// SIMATIC S7-200 SMART project (STEP 7-Micro/WIN SMART), CPU ST40

SYMBOL_TABLE Table 1
Item_detected    V0.0
Lid_at_place     V0.1
Base_at_place    V0.2
Part_leaving     V0.3
Start            V0.4
Reset            V0.5
Stop_            V0.6
Emergency_stop   V0.7
Auto             V1.0
FACTORY_IO_Running V1.1
X                VD100
Z                VD104
Lids_conveyor_1  Q2.0     // 0
Stop_blade_1     Q0.1
Lids_conveyor_2  Q2.1     // 0
Bases_conveyor_1 Q2.2     // 0
Stop_blade_2     Q0.4
Bases_conveyor_2 Q2.3     // 0
Grab             Q0.6
Start_light      Q0.7
Reset_light      Q1.0
Stop_light       Q1.1
Step_1_light     Q1.2
Step_2_light     Q1.3
Step_3_light     Q1.4
FACTOR_IO_Reset  Q1.5
Set_X            QD4
Set_Z            QD8
Counter          QD12
END_SYMBOL_TABLE

SYMBOL_TABLE System Symbols
Always_On        SM0.0    // Always ON
END_SYMBOL_TABLE

ORGANIZATION_BLOCK MAIN:OB1
TITLE=Program Comments
BEGIN
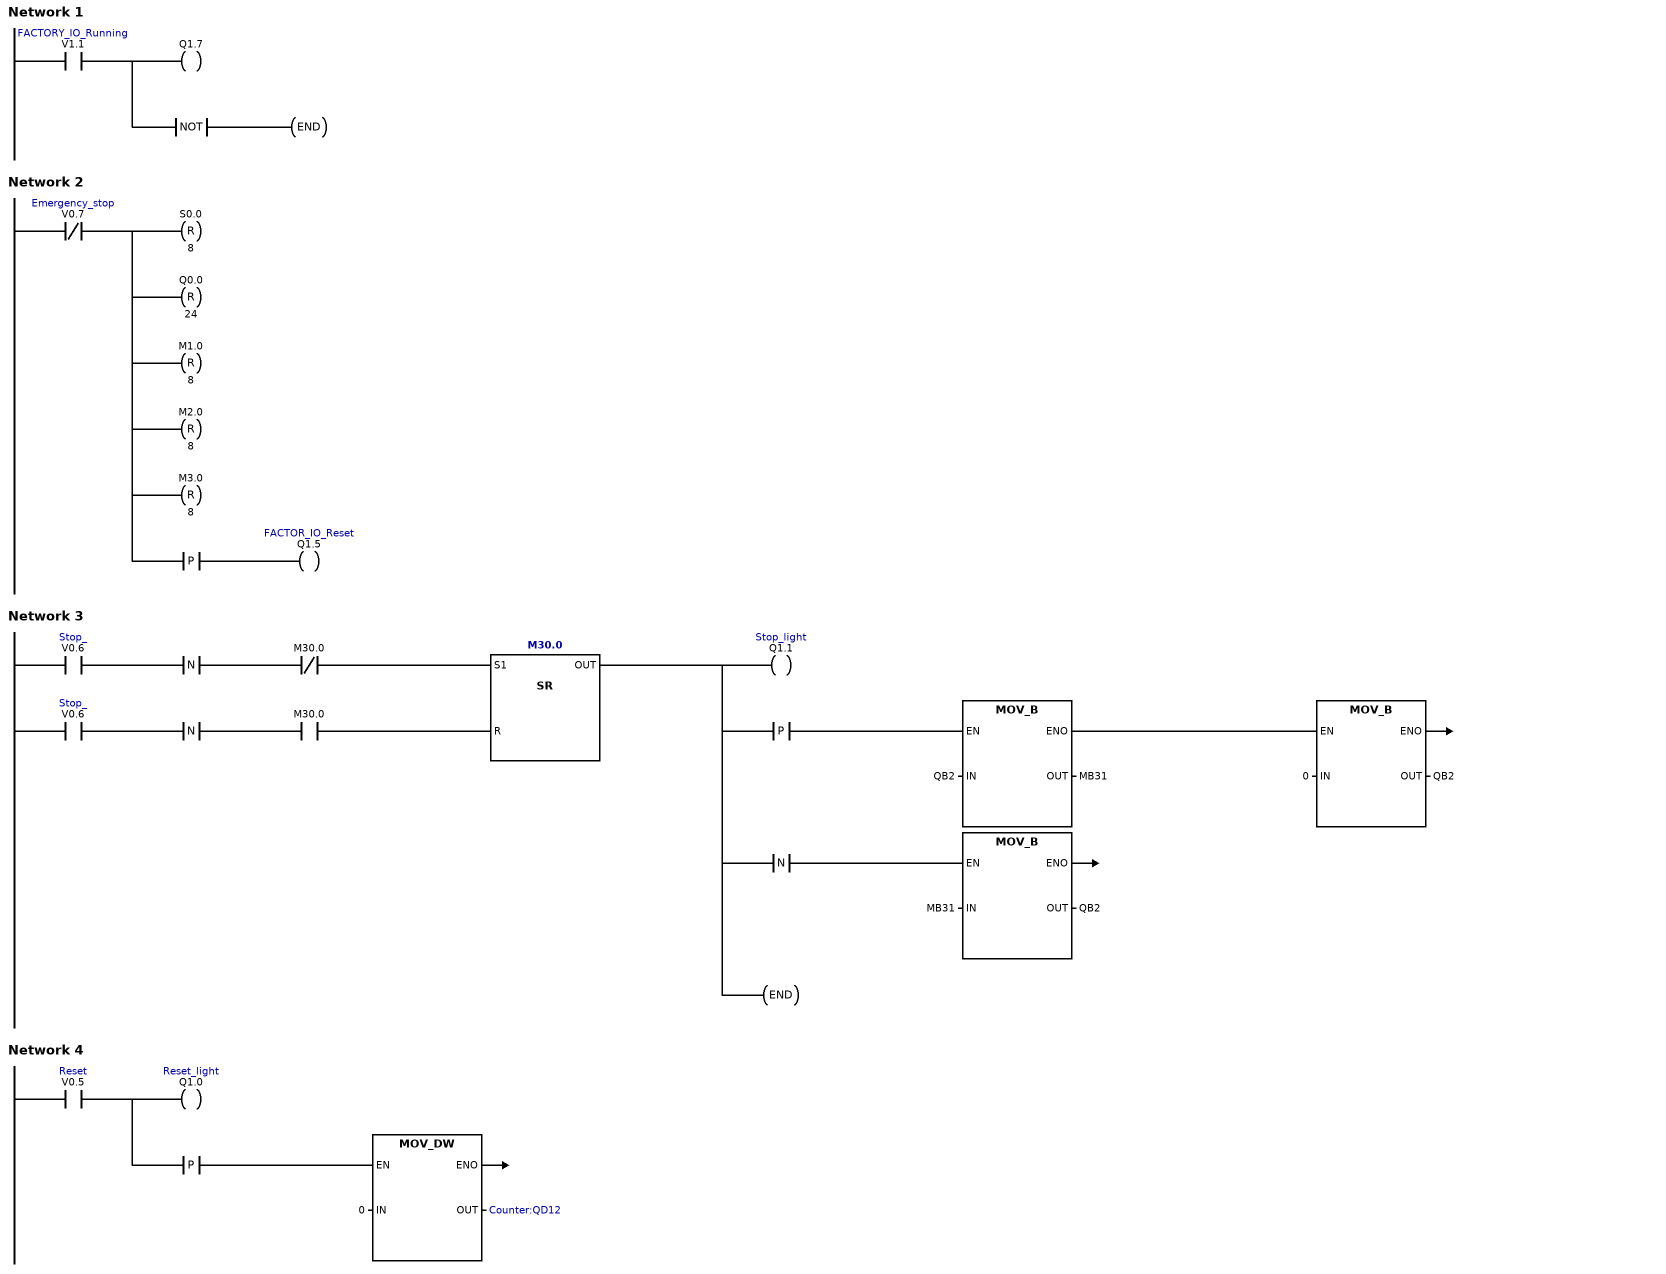
Network 1
LD     FACTORY_IO_Running:V1.1
=      Q1.7
NOT
END
Network 2
LDN    Emergency_stop:V0.7
R      S0.0, 8
R      Q0.0, 24
R      M1.0, 8
R      M2.0, 8
R      M3.0, 8
EU
=      FACTOR_IO_Reset:Q1.5
Network 3
LD     Stop_:V0.6
ED
AN     M30.0
LD     Stop_:V0.6
ED
A      M30.0
NOT
A      M30.0
OLD
=      M30.0
LPS
=      Stop_light:Q1.1
EU
MOVB   QB2, MB31
AENO
MOVB   0, QB2
LRD
ED
MOVB   MB31, QB2
LPP
END
Network 4
LD     Reset:V0.5
=      Reset_light:Q1.0
EU
MOVD   0, Counter:QD12
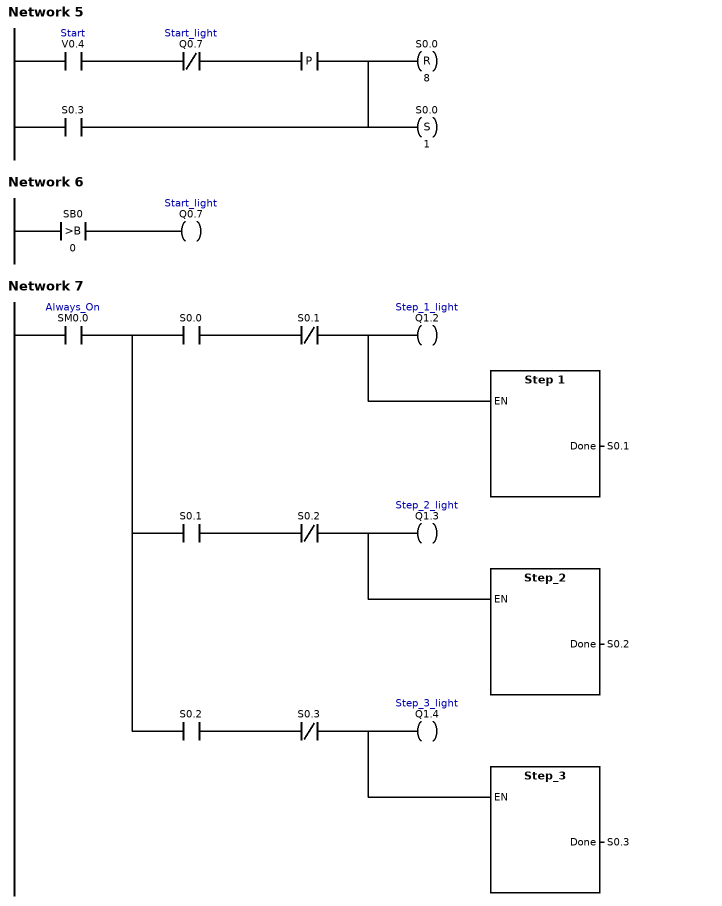
Network 5
LD     Start:V0.4
AN     Start_light:Q0.7
EU
O      S0.3
R      S0.0, 8
S      S0.0, 1
Network 6
LDB>   SB0, 0
=      Start_light:Q0.7
Network 7
LD     Always_On:SM0.0
LPS
A      S0.0
AN     S0.1
=      Step_1_light:Q1.2
CALL   Step 1:SBR1, S0.1
LRD
A      S0.1
AN     S0.2
=      Step_2_light:Q1.3
CALL   Step_2:SBR2, S0.2
LPP
A      S0.2
AN     S0.3
=      Step_3_light:Q1.4
CALL   Step_3:SBR3, S0.3
END_ORGANIZATION_BLOCK

SUBROUTINE_BLOCK Move:SBR0
TITLE=Subroutine Comments
VAR_INPUT
Set_X:REAL;	// LD0 
Set_Z:REAL;	// LD4 
END_VAR
VAR_OUTPUT
Done:BOOL;	// L8.0 
END_VAR
VAR
tmp:BOOL;	// L8.1 
tmp_x:REAL;	// LD9 
tmp_z:REAL;	// LD13 
END_VAR
BEGIN
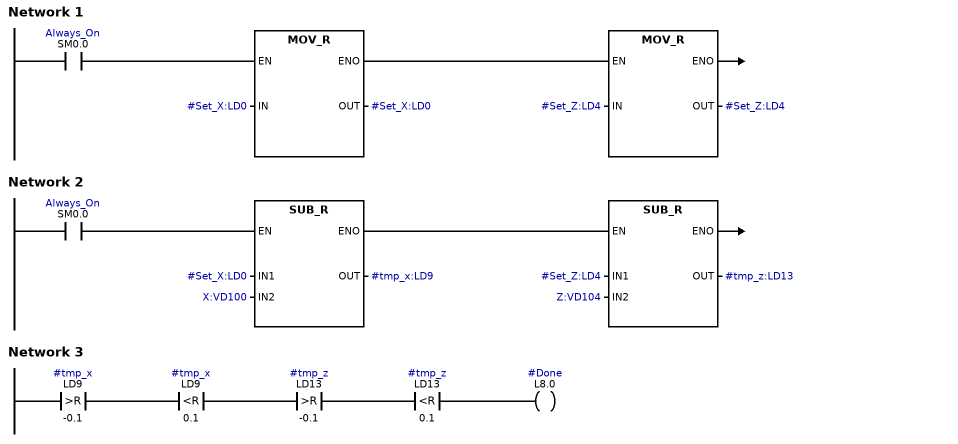
Network 1
LD     Always_On:SM0.0
MOVR   #Set_X:LD0, Set_X:QD4
AENO
MOVR   #Set_Z:LD4, Set_Z:QD8
Network 2
// (network saved uncompiled; LAD cells follow)
// row 0: c0 -| |- Always_On:SM0.0  c1 --  c2 [SUB_R EN:=power@row0, IN1:=#Set_X:LD0, IN2:=X:VD100, ENO=>power, OUT=>#tmp_x:LD9]  c3 --  c4 --  c5 [SUB_R EN:=power@row0, IN1:=#Set_Z:LD4, IN2:=Z:VD104, ENO=>power, OUT=>#tmp_z:LD13]  c6 ->
// row 1: c2 [box]  c5 [box]
Network 3
LDR>   #tmp_x:LD9, -0.1
AR<    #tmp_x:LD9, 0.1
AR>    #tmp_z:LD13, -0.1
AR<    #tmp_z:LD13, 0.1
=      #Done:L8.0
END_SUBROUTINE_BLOCK

SUBROUTINE_BLOCK Step 1:SBR1
TITLE=Subroutine Comments
VAR_OUTPUT
Done:BOOL;	// L0.0 
END_VAR
BEGIN
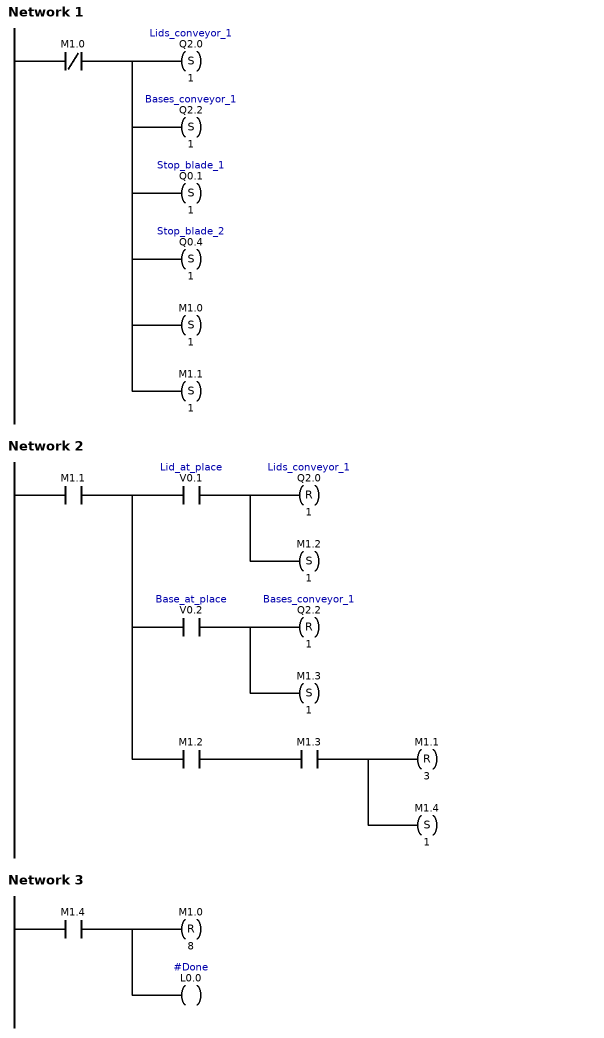
Network 1
LDN    M1.0
S      Lids_conveyor_1:Q2.0, 1
S      Bases_conveyor_1:Q2.2, 1
S      Stop_blade_1:Q0.1, 1
S      Stop_blade_2:Q0.4, 1
S      M1.0, 1
S      M1.1, 1
Network 2
LD     M1.1
LPS
A      Lid_at_place:V0.1
R      Lids_conveyor_1:Q2.0, 1
S      M1.2, 1
LRD
A      Base_at_place:V0.2
R      Bases_conveyor_1:Q2.2, 1
S      M1.3, 1
LPP
A      M1.2
A      M1.3
R      M1.1, 3
S      M1.4, 1
Network 3
LD     M1.4
R      M1.0, 8
=      #Done:L0.0
END_SUBROUTINE_BLOCK

SUBROUTINE_BLOCK Step_2:SBR2
TITLE=
VAR_OUTPUT
Done:BOOL;	// L0.0 
END_VAR
BEGIN
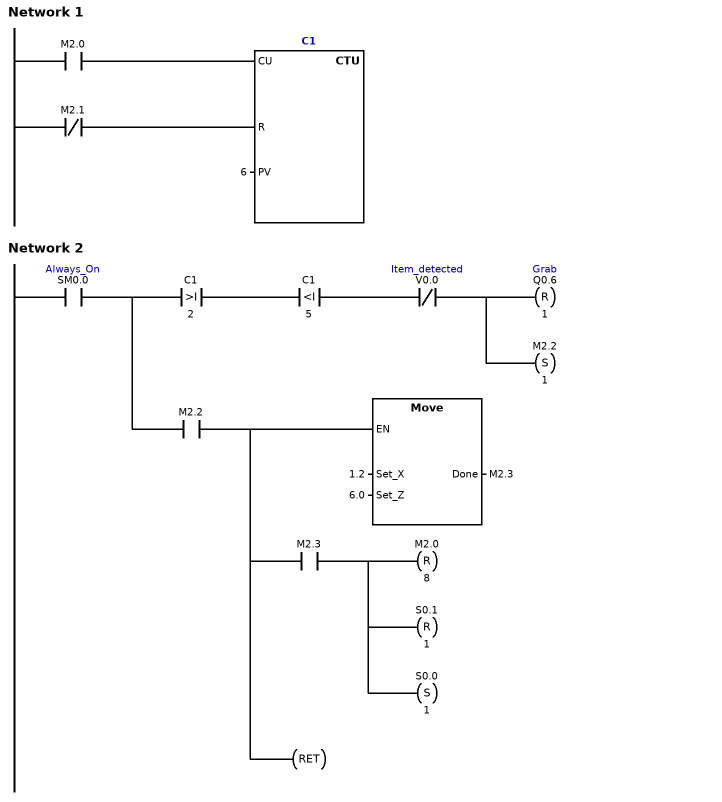
Network 1
LD     M2.0
LDN    M2.1
CTU    C1, 6
Network 2
LD     Always_On:SM0.0
LPS
AW>    C1, 2
AW<    C1, 5
AN     Item_detected:V0.0
R      Grab:Q0.6, 1
S      M2.2, 1
LPP
A      M2.2
LPS
CALL   Move:SBR0, 1.2, 6.0, M2.3
A      M2.3
R      M2.0, 8
R      S0.1, 1
S      S0.0, 1
LPP
CRET
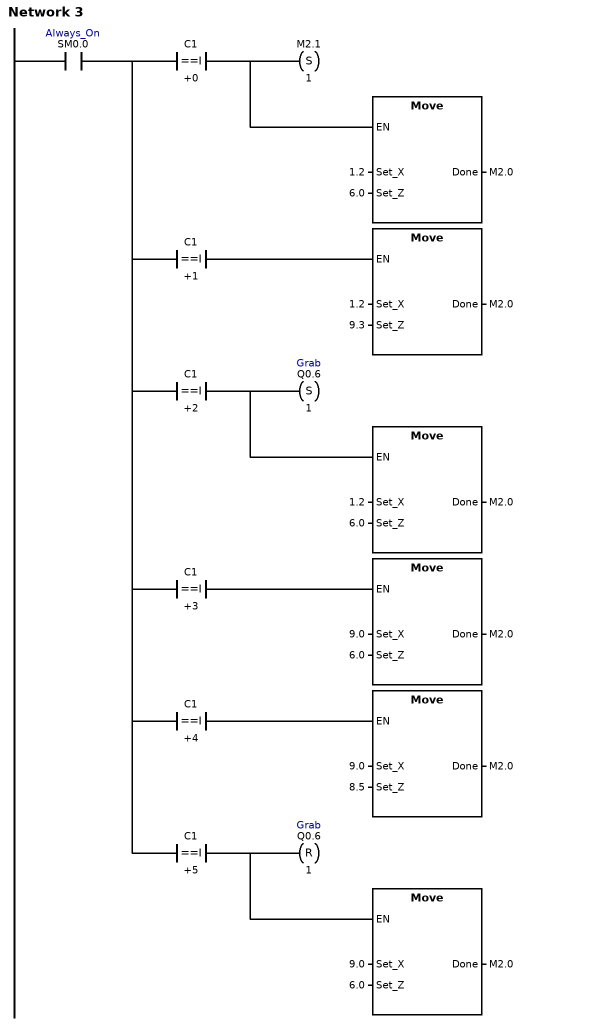
Network 3
LD     Always_On:SM0.0
LPS
AW=    C1, +0
S      M2.1, 1
CALL   Move:SBR0, 1.2, 6.0, M2.0
LRD
AW=    C1, +1
CALL   Move:SBR0, 1.2, 9.3, M2.0
LRD
AW=    C1, +2
S      Grab:Q0.6, 1
CALL   Move:SBR0, 1.2, 6.0, M2.0
LRD
LPS
AW=    C1, +3
CALL   Move:SBR0, 9.0, 6.0, M2.0
LPP
AW=    C1, +4
CALL   Move:SBR0, 9.0, 8.5, M2.0
LPP
AW=    C1, +5
R      Grab:Q0.6, 1
CALL   Move:SBR0, 9.0, 6.0, M2.0
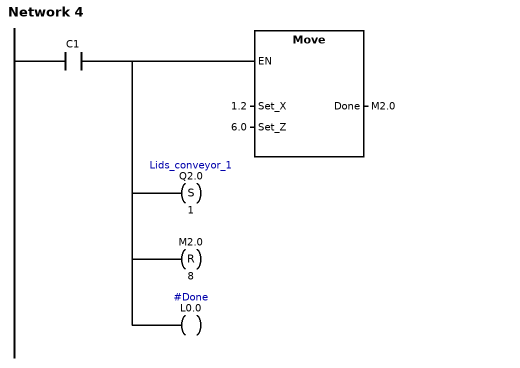
Network 4
LD     C1
CALL   Move:SBR0, 1.2, 6.0, M2.0
S      Lids_conveyor_1:Q2.0, 1
R      M2.0, 8
=      #Done:L0.0
END_SUBROUTINE_BLOCK

SUBROUTINE_BLOCK Step_3:SBR3
TITLE=Subroutine Comments
VAR_OUTPUT
Done:BOOL;	// L0.0 
END_VAR
BEGIN
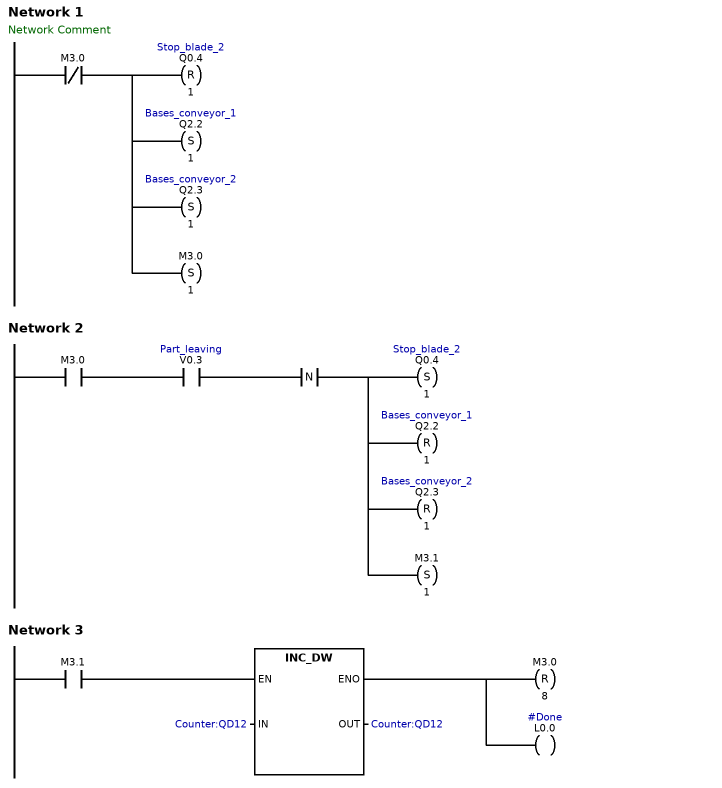
Network 1
// Network Comment
LDN    M3.0
R      Stop_blade_2:Q0.4, 1
S      Bases_conveyor_1:Q2.2, 1
S      Bases_conveyor_2:Q2.3, 1
S      M3.0, 1
Network 2
LD     M3.0
A      Part_leaving:V0.3
ED
S      Stop_blade_2:Q0.4, 1
R      Bases_conveyor_1:Q2.2, 1
R      Bases_conveyor_2:Q2.3, 1
S      M3.1, 1
Network 3
LD     M3.1
INCD   Counter:QD12
AENO
R      M3.0, 8
=      #Done:L0.0
END_SUBROUTINE_BLOCK
